// TIA Portal V17 export
// export: Created 2025-06-26T06:49:21.5073541Z, ExportSetting WithDefaults, DisplayName Totally Integrated Automation Portal, DisplayVersion V17 Update 8, DisplayName TIA Portal Openness, DisplayVersion V17 Update 8, DisplayName TIA Portal Version Control Interface, DisplayVersion V17, DisplayName STEP 7 Professional, DisplayVersion V17 Update 8, DisplayName STEP 7 Safety, DisplayVersion V17 Update 6, DisplayName WinCC Advanced, DisplayVersion V17 Update 8
DATA_BLOCK "DB_FromHB"   // DB100
{ S7_Optimized_Access := 'FALSE' }
VERSION : 0.1
// stored: AutoNumber false, DBAccessibleFromOPCUA true, IsOnlyStoredInLoadMemory false, IsWriteProtectedInAS false
   VAR
      CompressorMotorPower : Real;   // [kW]
      CompressorMotorSpeed : Real;   // [rpm]
      HBL_CT_524 : Real;   // [ppm]
      HBL_CT_538 : Real;   // [ppm]
      HBL_CT_615 : Real;   // [ppm]
      HBL_CT_620 : Real;   // [ppm]
      HBL_CT_643 : Real;   // [ppm]
      HBL_CT_673 : Real;   // [ppm]
      TemperatureLift : Real;   // [C]
      COP : Real;   // [1]
      HeatSinkHeatRate : Real;   // [kW]
      HeatboosterPerformance : Real;   // [%]
      WatchdogCounter : UInt;   // Liveness counter (free-running)
      RunningTimeHours : UInt;   // [h]
      RunningTimeMinutes : UInt;   // [min]
      RunningTimeSeconds : UInt;   // [s]
      HeatboosterState : UInt;   // 0 = Initialization, 1 = Offline, 2 = Standby, 3 = Prepare start, 4 = Start, 5 = Warmup, 6 = Run, 7 = Stop
      EmergencyStopStatus : Bool;   // 1 = E-stop ok, 0 = E-stop active
      AlarmActive : Bool;   // 1 = Common alarm active, 0 = Common alarm not active
      WarningActive : Bool;   // 1 = Common warning active, 0 = Common warning not active
      HBL_EC_01 : Bool;   // 1 = heaters on, 0 = heaters off
      HBL_EC_02 : Bool;   // 1 = heaters on, 0 = heaters off
      SSC_P_01 : Bool;   // 1 = pump running, 0 = pump off
      SSC_P_02 : Bool;   // 1 = pump running, 0 = pump off
      SSC_F_01 : Bool;   // 1 = fan running, 0 = fan off
      HBL_PZH_539 : Bool;   // 1 = switch active, 0 = switch not active
      HBL_HV_563 : Bool;
      HBL_HV_564 : Bool;
      HBL_HV_630 : Bool;
      HBL_HV_631 : Bool;
      HBL_HV_640_X1 : Bool;
      HBL_HV_640_X2 : Bool;
      HBL_HV_670_X1 : Bool;
      HBL_HV_670_X2 : Bool;
      HBL_HV_676 : Bool;
      CPC_HV_852_X1 : Bool;
      CPC_HV_852_X2 : Bool;
      HBL_HV_861_X1 : Bool;
      HBL_HV_861_X2 : Bool;
      CPC_LSH_870A : Bool;
      CPC_LSL_870B : Bool;
      CPC_PSH_874 : Bool;
      HBL_LSH_632 : Bool;
      HBL_LSL_633 : Bool;
      HBL_LS_644 : Bool;
      HBL_LS_674 : Bool;
      Spare615 : Bool;
      Spare616 : Bool;
      Spare617 : Bool;
      Alarms : Array[0..191] of Bool;   // 0 = no alarm, 1 = active or active unacknowledged alarm
      HBL_SC_03_A1 : Real;   // [rpm]
      HBL_SC_03_A2 : Real;   // [%]
      HBL_SC_03_A3 : Real;   // [kW]
      HBL_SC_01_A1 : Real;   // [rpm]
      HBL_SC_01_A2 : Real;   // [%]
      HBL_SC_01_A3 : Real;   // [kW]
      HBL_SC_02_A1 : Real;   // [rpm]
      HBL_SC_02_A2 : Real;   // [%]
      HBL_SC_02_A3 : Real;   // [kW]
      HBL_SC_10_A1 : Real;   // [rpm]
      HBL_SC_10_A2 : Real;   // [%]
      HBL_SC_10_A3 : Real;   // [kW]
      HBL_TT_18 : Real;   // [C]
      HBL_TT_03 : Real;   // [C]
      HBL_TT_21 : Real;   // [C]
      HBL_TT_22 : Real;   // [C]
      SSC_LT_01 : Real;
      SSC_PDT_01 : Real;
      SSC_PIT_01 : Real;
      SSC_TT_01 : Real;   // [C]
      SSC_TT_02 : Real;   // [C]
      SSC_TT_03 : Real;   // [C]
      SSC_TT_04 : Real;   // [C]
      HBL_TT_502 : Real;   // [C]
      HBL_PT_503 : Real;
      HBL_TT_504 : Real;   // [C]
      HBL_TT_505 : Real;   // [C]
      HBL_PT_506 : Real;
      HBL_LT_510 : Real;
      HBL_PT_511 : Real;
      HBL_TT_512 : Real;   // [C]
      HBL_HCV_514_A1 : Real;
      HBL_HCV_515_A1 : Real;
      HBL_TT_516 : Real;   // [C]
      HBL_PT_517 : Real;
      HBL_TT_518 : Real;   // [C]
      HBL_PT_519 : Real;
      HBL_TT_525 : Real;
      HBL_PT_526 : Real;
      HBL_FT_527 : Real;
      HBL_TT_530 : Real;
      HBL_PT_531 : Real;
      HBL_TT_532 : Real;
      HBL_TT_533 : Real;
      HBL_PT_534 : Real;
      HBL_AT_535 : Real;
      HBL_TT_16 : Real;
      HBL_TT_540 : Real;
      HBL_PT_541 : Real;
      HBL_TT_542 : Real;
      HBL_TT_543 : Real;
      HBL_PT_544 : Real;
      HBL_AT_545 : Real;
      HBL_TT_546 : Real;
      HBL_PT_547 : Real;
      HBL_HCV_548_A1 : Real;
      HBL_TT_17 : Real;
      HBL_PT_561 : Real;
      HBL_PT_562 : Real;
      HBL_FT_565 : Real;
      HBL_FT_566 : Real;
      HBL_TT_571 : Real;
      HBL_PT_572 : Real;
      HBL_TT_573 : Real;
      HBL_HCV_575_A1 : Real;
      HBL_HCV_576_A1 : Real;
      HBL_HCV_578_A1 : Real;
      HBL_PT_580 : Real;
      HBL_LIT_610 : Real;
      HBL_TT_611 : Real;
      HBL_PT_612 : Real;
      HBL_HCV_616_A1 : Real;
      HBL_PT_618 : Real;
      HBL_HCV_700_A1 : Real;
      HBL_PT_701 : Real;
      HBL_PT_702 : Real;
      HBL_PT_05 : Real;
      HBL_TT_23 : Real;
      HBL_TT_24 : Real;
      HBL_TT_25 : Real;
      HBL_TT_26 : Real;
      HBL_TT_27 : Real;
      CPC_CT_851 : Real;
      CPC_HCV_853_A1 : Real;
      CPC_PT_862 : Real;
      CPC_PT_865 : Real;
      CPC_TT_866 : Real;
      CPC_TT_871 : Real;
      CPC_PT_872 : Real;
      CPC_HCV_880_A1 : Real;
      HBL_HCV_900_A1 : Real;
      HBL_TT_901 : Real;
      HBL_PT_902 : Real;
      HBL_FT_903 : Real;
      HBL_CT_950 : Real;
      HBL_CT_951 : Real;
      HBL_PT_960 : Real;
      HBL_PT_961 : Real;
      CompressorVolumetricEfficiency : Real;
      CompressorIsentropicEfficiency : Real;
      CompressorMassFlow : Real;
      HeatSinkPinch : Real;
      HeatSinkMassFlow : Real;
      HeatSourceHeatRate : Real;
      HeatSourcePinch : Real;
      HeatSourceMassFlow : Real;
   END_VAR
BEGIN
END_DATA_BLOCK
